FUNCTION_BLOCK ABSTRACT FBA_SEQUENCE
VAR_IN_OUT
	AlarmRepository : FB_ALARM_REPOSITORY;
END_VAR
VAR_INPUT
END_VAR
VAR_OUTPUT
	Initialized : BOOL;
END_VAR
VAR
	_state : FB_STATE_MACHINE;
END_VAR

METHOD PUBLIC ABSTRACT Initialize : REFERENCE TO FBA_SEQUENCE
VAR_INPUT
END_VAR
END_METHOD

METHOD PUBLIC ABSTRACT Reset : REFERENCE TO FBA_SEQUENCE
VAR_INPUT
END_VAR
END_METHOD

END_FUNCTION_BLOCK

(* stored: Version 1.1.0.1, ProductVersion 3.1.4024.12
   POU FBA_SEQUENCE: Id {6b098270-d4d3-4b0a-9504-d01b905633b1}, SpecialFunc None
   Method Initialize: Id {106f4149-e459-4d74-a903-44f42b52a495}
   Method Reset: Id {dd4033d9-8b93-4ae0-879e-4986000482ac} *)
